{attribute addProperty BoxType "EL6690-0002-0000"}
{attribute addProperty Id "CycleTimerAT %I*ARRAY [0..2] OF USINT001ErrorCodeAT %I*BYTE812"}
{attribute addProperty CRC "2476952931"}
{attribute addProperty SizeInBites "8"}
{attribute addProperty SizeInBytes "1"}
TYPE Status_93A34D63 :
STRUCT
	{attribute addProperty Name "CycleTimer"}
	CycleTimer AT %I* : ARRAY [0..2] OF USINT;
	{attribute addProperty Name "ErrorCode"}
	ErrorCode AT %I* : BYTE;
END_STRUCT
END_TYPE

(* stored: Version 1.2.0.0, ProductVersion 3.1.4024.9
   DUT Status_93A34D63: Id {13bb806e-8e1e-4e84-9f32-71859ddbbcbd} *)
